// TIA Portal project "Ejercicio_Montacargas_26082026" (V13)

(* hardware
DEVICE "S7-1200 station_1"  S7-1200 Station
   slot 0: "Rack_0"  Rack  V1.0
   slot 1: "PLC_1"  CPU 1214C AC/DC/Rly  6ES7 214-1BE30-0XB0  V2.2
*)

// ===== PLC "PLC_1"  CPU 1214C AC/DC/Rly =====

VAR_GLOBAL   // PLC tag table "Tabla de variables estándar"
   "S1P" AT %I0.0 : Bool;
   "SPB" AT %I0.1 : Bool;
   "P1P" AT %I0.3 : Bool;
   "PPB" AT %I0.4 : Bool;
   "PSS" AT %I0.5 : Bool;
   "M_SUBE" AT %Q0.0 : Bool;
   "M_BAJA" AT %Q0.1 : Bool;
   "SSS" AT %I0.2 : Bool;
   "M0" AT %M10.0 : Bool;
   "M1" AT %M10.1 : Bool;
   "M2" AT %M10.2 : Bool;
   "M3" AT %M10.3 : Bool;
END_VAR

ORGANIZATION_BLOCK "Main"   // OB1, LAD, ProgramCycle
TITLE = "Main Program Sweep (Cycle)"
{ S7_Optimized_Access := 'FALSE' }
VERSION : 0.1
   VAR_TEMP   // added for the SCL form of the ladder/FBD networks
      _w1 : Bool;
   END_VAR
BEGIN

REGION Network 1
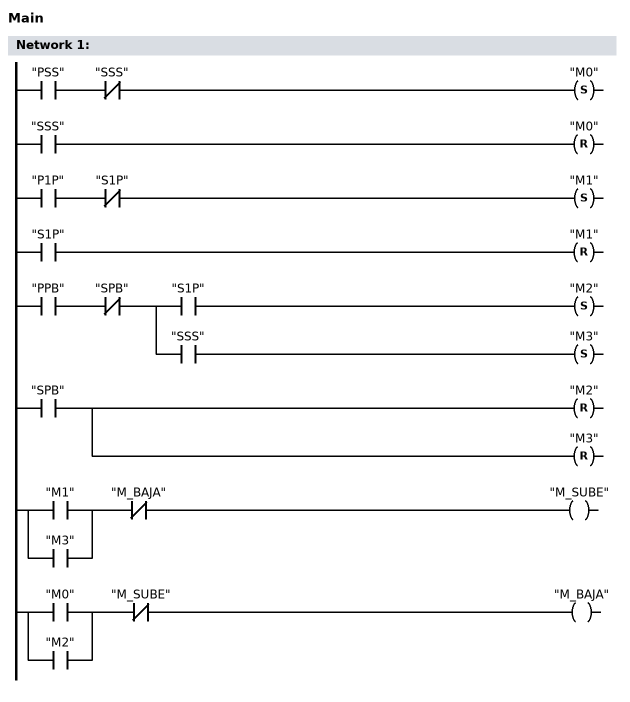
   RUNG wire#powerrail
      Contact( "PSS" )
      I_Contact( "SSS" )
      S_Coil( "M0" )
   END_RUNG
   RUNG wire#powerrail
      Contact( "SSS" )
      R_Coil( "M0" )
   END_RUNG
   RUNG wire#powerrail
      Contact( "P1P" )
      I_Contact( "S1P" )
      S_Coil( "M1" )
   END_RUNG
   RUNG wire#powerrail
      Contact( "S1P" )
      R_Coil( "M1" )
   END_RUNG
   RUNG wire#powerrail
      Contact( "PPB" )
      I_Contact( "SPB" )
      wire#w1
      Contact( "S1P" )
      S_Coil( "M2" )
   END_RUNG
   RUNG wire#w1
      Contact( "SSS" )
      S_Coil( "M3" )
   END_RUNG
   RUNG wire#powerrail
      Contact( "SPB" )
      wire#w2
      R_Coil( "M2" )
   END_RUNG
   RUNG wire#w2
      R_Coil( "M3" )
   END_RUNG
   RUNG wire#powerrail
      Contact( "M1" )
      wire#w3
      I_Contact( "M_BAJA" )
      Coil( "M_SUBE" )
   END_RUNG
   RUNG wire#powerrail
      Contact( "M3" )
   END_RUNG wire#w3
   RUNG wire#powerrail
      Contact( "M0" )
      wire#w4
      I_Contact( "M_SUBE" )
      Coil( "M_BAJA" )
   END_RUNG
   RUNG wire#powerrail
      Contact( "M2" )
   END_RUNG wire#w4
   // the same network as SCL:
   IF "PSS" AND NOT "SSS" THEN "M0" := TRUE; END_IF;
   IF "SSS" THEN "M0" := FALSE; END_IF;
   IF "P1P" AND NOT "S1P" THEN "M1" := TRUE; END_IF;
   IF "S1P" THEN "M1" := FALSE; END_IF;
   #_w1 := "PPB" AND NOT "SPB";
   IF #_w1 AND "S1P" THEN "M2" := TRUE; END_IF;
   IF #_w1 AND "SSS" THEN "M3" := TRUE; END_IF;
   IF "SPB" THEN
       "M2" := FALSE;
       "M3" := FALSE;
   END_IF;
   "M_SUBE" := ("M1" OR "M3") AND NOT "M_BAJA";
   "M_BAJA" := ("M0" OR "M2") AND NOT "M_SUBE";
END_REGION
END_ORGANIZATION_BLOCK